Universal Robots PolyScope program: send_robot_information.urp

Program send_robot_information (installation=default directory=/programs createdIn=5.2.0.61336 lastSavedIn=5.2.0.61336 robotSerialNumber=20185300040)
Calibrated DH parameters: a=[-0.000128, -0.221415, -0.194849, 0.000098, -0.000148, 0]; d=[0.152137, 33.879231, 13.968137, -47.716378, 0.085395, 0.092257]; alpha=[1.57105, 0.003021, -0.001826, 1.571145, -1.57192, 0]; deltaTheta=[0, 0.433042, -0.854582, 0.421536, 0.000002, 0]
BeforeStart
  var_1 := socket_open("10.0.47.225", 30002)
Robot Program (runOnlyOnce=false)
  Loop While (checkContinuously=false) expression=var_1≟ False
    var_1 := socket_open("10.0.47.225", 30002)
    Wait Sleep waitTime=0.5
  Script: socket_send_string("ask_me")
  Wait Sleep waitTime=0.5
  var_2 := socket_read_ascii_float(1)
  Wait Sleep waitTime=0.5
  If var_2[0]≠0
    Switch expression=var_2[1]
      Case (caseValue=1)
        pos := get_actual_tcp_pose()
        Script: socket_send_string(pos)
  var_1 := False
  Script: socket_close()
